FUNCTION_BLOCK FB_AutomaticControl
VAR_INPUT
	bEnable : BOOL;
	bActivateMotion : BOOL;
	bStopMotion : BOOL;
	stMotionReferenceGeneratorSettings : ST_MotionReferenceGeneratorSettings;
	stParam : ST_Parameters; 
END_VAR
VAR_OUTPUT
	fOutAutoTestPos : LREAL; 
	fOutAutoTestVel : LREAL; 
END_VAR
VAR
	fbClock : FB_Clock;	
	fbMotionReferenceGenerator : FB_MotionReferenceGenerator_limit;	
END_VAR

fbClock(
	bStart := bActivateMotion,
	bStop := bStopMotion,
	fCycleTime := stParam.fCyclicTime
);

fbMotionReferenceGenerator(
	bEnable := bEnable,
	stMotionReferenceGeneratorSettings := stMotionReferenceGeneratorSettings,
	fClock_s := fbClock.fTime
);

fOutAutoTestPos := fbMotionReferenceGenerator.fPositionReference_m;
fOutAutoTestVel := fbMotionReferenceGenerator.fVelocityReference_ms;

END_FUNCTION_BLOCK

(* stored: Version 1.1.0.1, ProductVersion 3.1.4024.9
   POU FB_AutomaticControl: Id {b543be1d-46f1-4ea5-ae35-9d7ea7728984}, SpecialFunc None *)
